Fanuc KAREL source: KT00728.KL

PROGRAM KT00728
%NOLOCKGROUP
VAR
  C1: CONFIG
  C2: CONFIG
  OUT: BOOLEAN
BEGIN
  C1.CFG_FLIP = TRUE
  C2.CFG_FLIP = FALSE
  C1.CFG_FLIP = TRUE
  C2.CFG_FLIP = FALSE
  OUT = UNINIT(C1)
END KT00728
